FUNCTION F_REAL_TO_STRING : STRING
VAR_INPUT
	rReal			: REAL;
	iPrecision		: INT;
END_VAR
VAR
	iTempInt		: DINT;
	iWholeNum		: DINT;
	iDecimal		: DINT;
	
	iAddZeros		: INT;
	
	sOut			: STRING;
	
	i				: INT;
END_VAR

IF RealIsNaN(rReal) THEN
	RETURN;
END_IF

iTempInt := REAL_TO_DINT(rReal * EXPT(10,ABS(iPrecision)));

iWholeNum	:= TRUNC(iTempInt / EXPT(10,ABS(iPrecision)));

iDecimal	:= iTempInt - LREAL_TO_DINT(iWholeNum * EXPT(10,ABS(iPrecision)));

sOut		:= CONCAT(DINT_TO_STRING(iWholeNum), '.');

IF iDecimal > 0 THEN
	iAddZeros	:= ABS(iPrecision) - DINT_TO_INT(TRUNC(LOG(iDecimal))) - 1;

	FOR i := 1 TO iAddZeros DO
		sOut	:= CONCAT(sOut,'0');
	END_FOR
	
	sOut	:= CONCAT(sOut, DINT_TO_STRING(iDecimal));
ELSE
	iAddZeros	:= ABS(iPrecision);

	FOR i := 1 TO iAddZeros DO
		sOut	:= CONCAT(sOut,'0');
	END_FOR
END_IF

F_REAL_TO_STRING	:= sOut;

END_FUNCTION

(* stored: Version 1.1.0.1, ProductVersion 3.1.4024.12
   POU F_REAL_TO_STRING: Id {27593807-da48-47d1-9404-780258f75522}, SpecialFunc None *)
